{attribute addProperty BoxType "EKM1101-0000-0016"}
{attribute addProperty Id "DiagBIT10.1251ErrorBIT10.1252Input_cycle_Counter_BIT_0BIT10.1253Input_cycle_Counter_BIT_1BIT10.1253TxPDO_StateBIT10.1257IDUSINT819"}
{attribute addProperty CRC "3179669839"}
{attribute addProperty SizeInBites "16"}
{attribute addProperty SizeInBytes "2"}
TYPE Status_BD85E94F :
STRUCT
	{attribute addProperty Name "Diag"}
	Diag : BIT;
	{attribute addProperty Name "Error"}
	Error : BIT;
	{attribute addProperty Name "Input_cycle_Counter"}
	Input_cycle_Counter_BIT_0 : BIT;
	{attribute addProperty Name "Input_cycle_Counter"}
	Input_cycle_Counter_BIT_1 : BIT;
	{attribute 'hide'}
	reserve_1_BIT_0 : BIT;
	{attribute 'hide'}
	reserve_1_BIT_1 : BIT;
	{attribute addProperty Name "TxPDO_State"}
	TxPDO_State : BIT;
	{attribute 'hide'}
	reserve_2 : BIT;
	{attribute addProperty Name "ID"}
	ID : USINT;
END_STRUCT
END_TYPE

(* stored: Version 1.2.0.0, ProductVersion 3.1.4024.9
   DUT Status_BD85E94F: Id {2592ea95-037e-46ab-9b33-999ad2fe74a5} *)
